// TwinCAT 3 PLC project Untitled1
// ProgramVersion: 3.1.4023.0
// libraries:
//   Tc2_Standard, * (Beckhoff Automation GmbH)
//   Tc2_System, * (Beckhoff Automation GmbH)
//   Tc3_Module, * (Beckhoff Automation GmbH)
// project tree:
//   DUTs/ A21ToolStorage.TcDUT (not stored), PositionMaterials.TcDUT (not stored)
//   DUTs/Enums/ A21.TcDUT, AirMode.TcDUT (not stored), Homing.TcDUT (not stored), SectionEnum.TcDUT (not stored), Surface.TcDUT, WoodBunk.TcDUT (not stored)
//   DUTs/Insertion/ AirSlider.TcPOU (not stored), PneumaticInsertion.TcPOU (not stored), SuctionPad.TcDUT, TeknicEIP.TcPOU (not stored)
//   DUTs/Machines/ Robot.TcPOU (not stored), StrapMachine.TcPOU (not stored)
//   DUTs/Material Holders/ MaterialStorage.TcPOU (not stored), WoodBunkTable.TcPOU (not stored)
//   GVLs/ GVL.TcGVL
//   / PlcTask.TcTTO
//   POUs/ MAIN.TcPOU
// real-time tasks:
//   TASK PlcTask: cycle T#10ms, priority 20, ADS port 350
//   TASK PlcTask1: cycle T#10ms, priority 21, ADS port 351

CONFIGURATION Untitled1
    RESOURCE PLC ON TwinCAT3
        TASK PlcTask(INTERVAL := T#10ms, PRIORITY := 21);
        PROGRAM MAIN WITH PlcTask : MAIN;
    END_RESOURCE
END_CONFIGURATION

// ---- DUTs/Enums/A21.TcDUT
{attribute 'qualified_only'}
{attribute 'strict'}
{attribute 'to_string'}
TYPE A21 :
(
	IDLE,
	STAGE_BUNK,
	REMOVE_BUNK_FROM_STAGE,
	
	LOAD_BUNK_TO_TOP := 4,
	LOAD_BUNK_TO_SIDE,
	LOAD_BUNK_TO_BOTTOM,
	REMOVE_BUNK_FROM_TOP,
	REMOVE_BUNK_FROM_SIDE,
	REMOVE_BUNK_FROM_BOTTOM,
	
	GET_CHIPBOARD_FROM_SKID := 11,
	REMOVE_CHIPBOARD_FROM_TOOL,
	PLACE_CHIPBOARD_TO_TOP,
	PLACE_CHIPBOARD_TO_BOTTOM,
	REMOVE_CHIPBOARD_TOP,
	REMOVE_CHIPBOARD_BOTTOM,
	
	FIX_CHIPBOARD_ORIENTATION := 19,
	
	//testing only
	MOVE_HOME := 21,
	MOVE_POSITION1,
	MOVE_POSITION2,
	MOVE_UP,
	MOVE_DOWN,
	
	DIRECT_BUNK_TO_TOP := 27,
	DIRECT_BUNK_TO_SIDE,
	DIRECT_BUNK_TO_BOTTOM,
	
	INSPECT_BUNK := 31,
	INSPECT_CHIPBOARD,
	
	TOOL_CHANGE_BUNK := 34,
	TOOL_CHANGE_CHIPBOARD,
	
	size
);
END_TYPE

// ---- DUTs/Enums/Surface.TcDUT
{attribute 'qualified_only'}
{attribute 'strict'}
TYPE Surface :
(
	TOP := 1,
	LEFT,
	RIGHT,
	BOTTOM,
	TOP_LEFT,
	TOP_RIGHT,
	BOTTOM_LEFT,
	BOTTOM_RIGHT,
	
	size
)BYTE;
END_TYPE

// ---- DUTs/Insertion/SuctionPad.TcDUT
TYPE SuctionPad :
STRUCT
	enableOut AT %Q* : BOOL;
	enableIn AT %I* : BOOL;
END_STRUCT
END_TYPE

// ---- GVLs/GVL.TcGVL
{attribute 'qualified_only'}
VAR_GLOBAL CONSTANT
	maxPairs : USINT := 16;
	initArraySize : USINT := 4;
	maxQueue : INT := 16;
	
	nullPos : REAL := -1;
	
	numMaterials : INT := 32;
	conveyorLength : REAL := 0;
	precisionTolerance : REAL := 0.05 * 25.4;
END_VAR
VAR_GLOBAL
	
END_VAR

// ---- POUs/MAIN.TcPOU
PROGRAM MAIN
VAR_INPUT
	execute : BOOL;
	manualMode : BOOL;
END_VAR
VAR_OUTPUT
	robotLeft, robotRight : Robot;
	
	stagingTableLeft, stagingTableRight : WoodBunkTable;
	magazineLeft, magazineRight : MaterialStorage;
	
	strapper : StrapMachine;
	
	insertionLeft, insertionRight : PneumaticInsertion;	
	insertionBottom : TeknicEIP;
	topSuction : ARRAY[1..3] OF SuctionPad;
	leftSuction, rightSuction : ARRAY[1..4] OF SuctionPad;
	bottomSuction : ARRAY[1..2] OF SuctionPad;
	
	toolStorageLeft : A21ToolStorage;
	toolStorageRight : A21ToolStorage;
	
	stagingTemplateLeft, stagingTemplateRight : WoodBunkTable;
END_VAR
VAR
	robotLeftOutputs, robotRightOutputs : ARRAY[1..50] OF INT;
	demoPair : PositionMaterials;
	demoHeight : REAL := 600; //600mm, 60cm
	
	sectionID : SectionEnum := SectionEnum.WOOD_BUNK;
	
	step : (IDLE, STAGING, LOADING, PUSH, STRAP, RELEASE, DONE);
	ready : BOOL;
	
	loadSet : INT;
	loadStepLeft, loadStepRight : INT;
	
	stageSet : INT;	
	stageStepLeft, stageStepRight : INT;
	iStagingSlotLeft, iStagingSlotRight : INT;
END_VAR
VAR CONSTANT
	COMPLETE : INT := 1050;
END_VAR

demoPair.position := 0;
demoPair.top := 'WDW20';
demoPair.left := 'WDS14';
demoPair.right := 'WDS14';
demoPair.bottom := 'WDB20';

setup();
hardwareLadder();

IF NOT ready THEN
	ready :=
		insertionLeft.homingSequence() AND
		insertionRight.homingSequence() AND
		insertionBottom.homingSequence();
END_IF


CASE step OF
	IDLE:
		IF execute THEN
			execute := FALSE;
			step := STAGING;
		END_IF
		
	STAGING:
		IF stage() THEN
			IF manualMode AND_THEN NOT execute THEN
				RETURN;
			END_IF
			
			step := LOADING;
		END_IF
	
	LOADING:
		IF load(pair := demoPair) THEN
			IF manualMode AND_THEN NOT execute THEN
				RETURN;
			END_IF
		
			step := STRAP;
		END_IF
		
	PUSH:
		insertionBottom.traverse(direction := FALSE);
		IF NOT insertionLeft.alignTarget(demoHeight/2) OR insertionRight.alignTarget(demoHeight/2) THEN
			RETURN;
		END_IF
		
		insertionBottom.traverse(direction := FALSE);
		insertionLeft.press();
		insertionRight.press();
		
		IF insertionBottom.contact AND insertionLeft.contact AND insertionRight.contact THEN
			step := STRAP;
		END_IF
		
	STRAP:
		IF strapper.ready OR (NOT strapper.busy AND NOT strapper.error) THEN
			strapper.strap();
		END_IF
		
		IF strapper.done THEN
			IF manualMode AND_THEN NOT execute THEN
				RETURN;
			END_IF
			
			step := RELEASE;
		END_IF
		
	RELEASE: //release command
		MEMSET(ADR(topSuction), 0, SIZEOF(topSuction));
		MEMSET(ADR(leftSuction), 0, SIZEOF(leftSuction));
		MEMSET(ADR(rightSuction), 0, SIZEOF(rightSuction));
		MEMSET(ADR(bottomSuction), 0, SIZEOF(bottomSuction));
		
		IF NOT insertionLeft.home THEN
			insertionLeft.alignTarget(0);
			insertionLeft.release();
		END_IF
		
		IF NOT insertionRight.home THEN
			insertionRight.alignTarget(0);
			insertionRight.release();
		END_IF
		
		IF insertionLeft.home AND insertionRight.home THEN
			IF manualMode AND_THEN NOT execute THEN
				RETURN;
			END_IF
			
			step := COMPLETE;
		END_IF
	
	COMPLETE:
		//reset everything
		step := IDLE;
		
END_CASE

METHOD changeRobotsEOAT : BOOL
VAR_INPUT
END_VAR
IF robotLeft.tool <> sectionID THEN
	MEMSET(ADR(robotLeftOutputs), 0, SIZEOF(robotLeftOutputs));
	robotLeftOutputs[1] := A21.TOOL_CHANGE_CHIPBOARD;
	robotLeft.setParamsAndWait(robotLeftOutputs);
END_IF

IF robotRight.tool <> sectionID THEN
	MEMSET(ADR(robotRightOutputs), 0, SIZEOF(robotRightOutputs));
	robotRightOutputs[1] := A21.TOOL_CHANGE_CHIPBOARD;
	robotRight.setParamsAndWait(robotRightOutputs);
END_IF

changeRobotsEOAT := robotLeft.tool = sectionID AND robotRight.tool = sectionID;
END_METHOD

METHOD PROTECTED createStagingTemplate : BOOL
VAR
	remainingMaterial : STRING;
	splitMaterial : STRING;
	
	i : INT;
END_VAR
stagingTemplateLeft.autofill(demoPair.top);
stagingTemplateLeft.autofill(demoPair.left);

stagingTemplateRight.autofill(demoPair.right);
stagingTemplateRight.autofill(demoPair.bottom);

createStagingTemplate := TRUE;

(*
FOR i:=0 TO GVL.maxPairs BY 1 DO //iterate through all pairs and autofill the template
	//LEFT TABLE
	remainingMaterial := materialsArr[i].top;
	WHILE FIND(remainingMaterial, '_') > 0 DO //until no underscore found
		splitCombinedMaterials(remainingMaterial, splitMaterial);
		stagingTemplateLeft.autofill(splitMaterial);
	END_WHILE
	stagingTemplateLeft.autofill(remainingMaterial);
	
	remainingMaterial := materialsArr[i].left;
	WHILE FIND(remainingMaterial, '_') > 0 DO
		splitCombinedMaterials(remainingMaterial, splitMaterial);
		stagingTemplateLeft.autofill(splitMaterial);
	END_WHILE
	stagingTemplateLeft.autofill(remainingMaterial);
	
	//RIGHT TABLE
	remainingMaterial := materialsArr[i].right;
	WHILE FIND(remainingMaterial, '_') > 0 DO
		splitCombinedMaterials(remainingMaterial, splitMaterial);
		stagingTemplateRight.autofill(splitMaterial);
	END_WHILE
	stagingTemplateRight.autofill(remainingMaterial);
	
	remainingMaterial := materialsArr[i].bottom;
	WHILE FIND(remainingMaterial, '_') > 0 DO
		splitCombinedMaterials(remainingMaterial, splitMaterial);
		stagingTemplateRight.autofill(splitMaterial);
	END_WHILE
	stagingTemplateRight.autofill(remainingMaterial);
END_FOR
createStagingTemplate := TRUE;
*)
END_METHOD

METHOD hardwareCall : BOOL
robotLeft();
robotRight();

stagingTableLeft();
stagingTableRight();

magazineLeft();
magazineRight();

strapper();

insertionLeft();
insertionRight();
insertionBottom();

stagingTemplateLeft();
stagingTemplateRight();
END_METHOD

METHOD hardwareLadder : BOOL
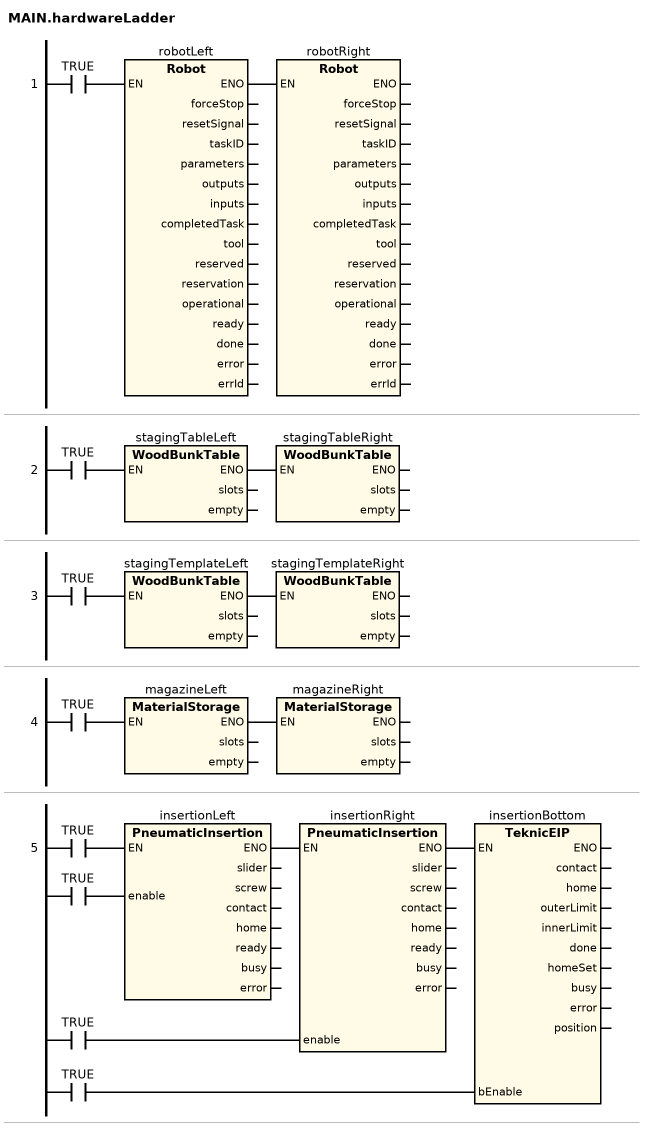
// NETWORK 1
robotLeft(); // Robot
robotRight(); // Robot

// NETWORK 2
stagingTableLeft(); // WoodBunkTable
stagingTableRight(); // WoodBunkTable

// NETWORK 3
stagingTemplateLeft(); // WoodBunkTable
stagingTemplateRight(); // WoodBunkTable

// NETWORK 4
magazineLeft(); // MaterialStorage
magazineRight(); // MaterialStorage

// NETWORK 5
insertionLeft(enable := TRUE); // PneumaticInsertion
insertionRight(enable := TRUE); // PneumaticInsertion
insertionBottom(bEnable := TRUE); // TeknicEIP
END_METHOD

METHOD PROTECTED load : BOOL
VAR_INPUT
	pair : REFERENCE TO PositionMaterials;
END_VAR
VAR_OUTPUT
	error : BOOL;
END_VAR
IF NOT robotLeft.operational OR NOT robotLeft.operational THEN
	error := TRUE;
	RETURN;
END_IF

IF NOT (robotLeft.reserve(sectionID) AND robotRight.reserve(sectionID)) THEN
	RETURN;
END_IF

IF NOT (robotLeft.tool = sectionID AND robotRight.tool = sectionID) THEN //robots have wrong tool
	changeRobotsEOAT(); //wait for robots to finish changing tools
	RETURN;
END_IF


CASE loadSet OF
	0: //top and bottom
		IF 
			loadingSequence(
				actingRobot:= robotLeft, 
				robotOutputs:= robotLeftOutputs, 
				stagingTable:= stagingTableLeft, 
				loadStep:= loadStepLeft, 
				suctions:= topSuction,
				surfaceID:= Surface.TOP, 
				material:= pair.top, 
				fail=> )
			AND
			loadingSequence(
				actingRobot:= robotRight, 
				robotOutputs:= robotRightOutputs, 
				stagingTable:= stagingTableRight, 
				loadStep:= loadStepRight, 
				suctions:= bottomSuction,
				surfaceID:= Surface.BOTTOM, 
				material:= pair.bottom, 
				fail=> )
		THEN
			loadStepLeft := loadStepRight := 0;
			loadSet := 10;
		END_IF
		
	10: //sides
		IF
			loadingSequence(
				actingRobot:= robotLeft, 
				robotOutputs:= robotLeftOutputs, 
				stagingTable:= stagingTableLeft, 
				loadStep:= loadStepLeft, 
				suctions:= leftSuction,
				surfaceID:= Surface.LEFT, 
				material:= pair.left, 
				fail=> )
			AND
			loadingSequence(
				actingRobot:= robotRight, 
				robotOutputs:= robotRightOutputs, 
				stagingTable:= stagingTableRight, 
				loadStep:= loadStepRight, 
				suctions:= rightSuction,
				surfaceID:= Surface.RIGHT, 
				material:= pair.right, 
				fail=> )
		THEN
			loadStepLeft := loadStepRight := 0;
			loadSet := COMPLETE;
		END_IF
		
	COMPLETE:
		loadSet := 0;
		loadStepLeft := loadStepRight := 0;
		
		robotLeft.release(sectionID);
		robotRight.release(sectionID);
		
		load := TRUE;
END_CASE
END_METHOD

METHOD loadingSequence : BOOL
VAR_IN_OUT
	actingRobot : Robot;
	robotOutputs : ARRAY[1..50] OF INT;
	stagingTable : WoodBunkTable;
	suctions : ARRAY[*] OF SuctionPad;
	loadStep : INT;
END_VAR
VAR_INPUT
	surfaceID : Surface;
	material : STRING;
END_VAR
VAR_OUTPUT
	fail : BOOL;
END_VAR
VAR
	slot : INT;
	i : DINT;
END_VAR
VAR
	suctionArr : POINTER TO SuctionPad;
	firstSuction : INT := 1;
	lastSuction : INT;
END_VAR
IF material = '' THEN
	loadingSequence := TRUE;
	RETURN;
END_IF

CASE loadStep OF
	0:
		IF NOT stagingTable.findSlot(materialID := material, atSlot => slot) THEN
			fail := TRUE;
			RETURN;
		END_IF
		
		MEMSET(ADR(robotOutputs), 0, SIZEOF(robotOutputs));
		CASE surfaceID OF
			Surface.TOP: 					robotOutputs[1] := A21.LOAD_BUNK_TO_TOP;
			Surface.LEFT, Surface.RIGHT: 	robotOutputs[1] := A21.LOAD_BUNK_TO_SIDE;
			Surface.BOTTOM: 				robotOutputs[1] := A21.LOAD_BUNK_TO_BOTTOM;
		END_CASE
		robotOutputs[2] := slot;
		
		IF actingRobot.setParamsAndWait(robotOutputs) THEN
			loadStep := COMPLETE;
		END_IF
		
	COMPLETE:
		FOR i:=LOWER_BOUND(suctions, 1) TO UPPER_BOUND(suctions, 1) BY 1 DO
			suctions[i].enableOut := TRUE;
		END_FOR
		
		actingRobot.release(sectionID);
		loadingSequence := TRUE;
		
END_CASE
END_METHOD

METHOD PRIVATE setup : BOOL
VAR
	iWoodBunkSlot : WoodBunk := 1;
	
	slotsArr : ARRAY[1..GVL.maxQueue] OF STRING;
	
	i : INT;
END_VAR
FOR iWoodBunkSlot:=1 TO WoodBunk.size-1 BY 1 DO
	slotsArr[iWoodBunkSlot] := TO_STRING(iWoodBunkSlot);
END_FOR
magazineLeft.setupSlots(slotsArr);
magazineRight.setupSlots(slotsArr);


insertionLeft.enable := insertionRight.enable := insertionBottom.bEnable := TRUE;

setup := TRUE;
END_METHOD

METHOD stage : BOOL
//robot reservation needs to be constantly checked so it is not in the state machine
IF NOT (robotLeft.reserve(sectionID) AND robotRight.reserve(sectionID)) THEN
	RETURN;
END_IF

IF NOT (robotLeft.tool = sectionID AND robotRight.tool = sectionID) THEN //robots have wrong tool
	changeRobotsEOAT(); //wait for robots to finish changing tools
	RETURN;
END_IF

CASE stageSet OF
	0: //create staging template
		IF createStagingTemplate() THEN
			step := 10;
		END_IF
	
	10: //staging sequence
		IF
			stagingSequence(
				template:= stagingTemplateLeft, 
				magazine:= magazineLeft, 
				table:= stagingTableLeft, 
				actingStagingSlot:= iStagingSlotLeft,
				actingRobot:= robotLeft, 
				robotOutputs:= robotLeftOutputs,
				actingStep:= stageStepLeft, 
				fail=> )
				
			AND
			stagingSequence(
				template:= stagingTemplateRight, 
				magazine:= magazineRight, 
				table:= stagingTableRight, 
				actingStagingSlot:= iStagingSlotRight,
				actingRobot:= robotRight, 
				robotOutputs:= robotRightOutputs,
				actingStep:= stageStepRight, 
				fail=> )
		THEN
			stageStepLeft := stageStepRight := 0;
			iStagingSlotLeft := iStagingSlotRight := 0;
			
			stageSet := COMPLETE;
		END_IF
		
	COMPLETE:
		stageSet := 0;
		stageStepLeft := stageStepRight := 0;
		
		robotLeft.release(sectionID);
		robotRight.release(sectionID);
		
		stage := TRUE;
		
END_CASE
END_METHOD

METHOD stageLeft : BOOL
VAR_IN_OUT
	template : WoodBunkTable;
	magazine : MaterialStorage;
	table : WoodBunkTable;
	actingStagingSlot : INT;
	actingRobot : Robot;
	robotOutputs : ARRAY[1..50] OF INT;
	actingStep : INT;
END_VAR
VAR_OUTPUT
	fail : BOOL;
END_VAR
VAR
	finished : BOOL;
	
	slot : INT;
	templateArr : POINTER TO STRING;
	//iSlot : REFERENCE TO INT; 
END_VAR
VAR CONSTANT
	WIP : INT := 0;
	PASSED : INT := 1;
	FAILED : INT := 2;
END_VAR
(*
IF table.isFull() OR actingStagingSlot > 10 THEN
	stageLeft := TRUE;
	RETURN;
END_IF

templateArr := template.getSlotsAsArray();

//follow the template as is
IF NOT magazine.findSlot(materialID:= templateArr[actingStagingSlot], atSlot => slot) THEN
	fail := TRUE;
	RETURN;
END_IF

IF actingStep > 0 THEN
	finished := actingRobot.setParamsAndWait(robotOutputs);
END_IF

CASE actingStep OF		
	0:
		IF actingRobot.inputs[5].10 THEN //in position for inspection
			robotOutputs[4] := PASSED;
			actingStep := 30;
		END_IF
		
	COMPLETE:
		IF finished THEN
			actingStep := 0;
		END_IF
END_CASE
*)
END_METHOD

METHOD stageRight : BOOL
VAR_IN_OUT
	template : WoodBunkTable;
	magazine : MaterialStorage;
	table : WoodBunkTable;
	actingStagingSlot : INT;
	actingRobot : Robot;
	actingStep : INT;
END_VAR
VAR_INPUT
	camera : INT;
END_VAR
VAR_OUTPUT
	fail : BOOL;
END_VAR
VAR
	finished : BOOL;
	robotOutputs : POINTER TO INT;
	
	slot : INT;
	templateArr : POINTER TO STRING;
	
END_VAR
(*
IF table.isFull() OR actingStagingSlot > 10 THEN
	stageRight := TRUE;
	RETURN;
END_IF

templateArr := template.getSlotsAsArray();

//follow the template as is
IF NOT magazine.findSlot(materialID:= templateArr[actingStagingSlot], atSlot => slot) THEN
	fail := TRUE;
	RETURN;
END_IF

IF actingStep > 0 THEN
	finished := actingRobot.setCommandAndWait(A21.STAGE_BUNK, slot, actingStagingSlot, 0);
END_IF

CASE actingStep OF
	0: //command
		IF actingRobot.inputs[5].10 THEN
			actingStep := 10;
		END_IF
		
	10: //send inspection data
		tempInspectionSuite.frame.MaterialID := templateArr[actingStagingSlot];
		tempInspectionSuite.frame.CheckFor := 'ORIENTATION';
		tempInspectionSuite.frame.CameraNumber := camera;
	
		CreateJsonDocumentAuto(
			visionFrameData:= tempInspectionSuite.frame, 
			jsonDocument=> tempInspectionSuite.json);
		
		MEMCPY( //data = json
			ADR(tempInspectionSuite.data), 
			ADR(tempInspectionSuite.json), 
			MIN( SIZEOF(tempInspectionSuite.data), SIZEOF(tempInspectionSuite.json) ));
			
		TcpServer1Vision.queue(tempInspectionSuite.data);
		
		actingStep := 20;
	
	20: //fetch inspection data and parse
		actingRobot.setCommandAndWait(A21.STAGE_BUNK, slot, actingStagingSlot, 0);
		robotOutputs[11] := 0;
		
		IF NOT FrameIsValid(actingFrame) THEN
			RETURN;
		END_IF
		
		IF actingFrame.SuccessFlag = 1 THEN
			robotOutputs[11] := 1;
		ELSE
			robotOutputs[11] := 2;
		END_IF
		step := 30;
		
	30: //finish command
		IF finished THEN
			IF actingFrame.SuccessFlag = 1 THEN
				actingStagingSlot := actingStagingSlot + 1;
			END_IF
			
			actingStep := 0; //stage next
		END_IF
		
END_CASE
*)
END_METHOD

METHOD stagingSequence : BOOL
VAR_IN_OUT
	template : WoodBunkTable;
	magazine : MaterialStorage;
	table : WoodBunkTable;
	actingStagingSlot : INT;
	actingRobot : Robot;
	robotOutputs : ARRAY[1..50] OF INT;
	actingStep : INT;
END_VAR
VAR_OUTPUT
	fail : BOOL;
END_VAR
VAR
	finished : BOOL;
	slot : INT;
	templateArr : POINTER TO STRING;
END_VAR
VAR CONSTANT
	WIP : INT := 0;
	PASSED : INT := 1;
	FAILED : INT := 2;
END_VAR
IF
	//table.isFull() OR actingStagingSlot > 10 OR
	MEMCMP(ADR(table.slots), templateArr, SIZEOF(table.slots)) = 0
	//MEMCMP(table.getSlotsAsArray(), templateArr, SIZEOF(templateArr)) = 0
THEN
	stagingSequence := TRUE;
	RETURN;
END_IF

templateArr := ADR(template.slots); // := template.getSlotsAsArray();

//follow the template as is
IF NOT magazine.findSlot(materialID:= templateArr[actingStagingSlot], atSlot => slot) THEN
	fail := TRUE;
	RETURN;
END_IF

IF actingStep > 0 THEN
	finished := actingRobot.setParamsAndWait(robotOutputs);
END_IF

CASE actingStep OF		
	0:
		IF actingRobot.inputs[5].10 THEN //in position for inspection
			robotOutputs[4] := PASSED;
			actingStep := 30;
		END_IF
		
	30:
		IF finished THEN
			actingStep := COMPLETE;
		END_IF
		
	COMPLETE:
		MEMSET(ADR(robotOutputs), 0, SIZEOF(robotOutputs));
		actingStagingSlot := actingStagingSlot + 1;
		//stagingSequence := TRUE;
END_CASE
END_METHOD

END_PROGRAM
